Fanuc TP program (LS listing): _bgl_btn_pick.ls

/PROG  _BGL_BTN_PICK
/ATTR
OWNER		= MNEDITOR;
COMMENT		= "";
PROG_SIZE	= 225;
CREATE		= DATE 00-01-12  TIME 18:35:34;
MODIFIED	= DATE 00-01-12  TIME 18:35:34;
FILE_NAME	= ;
VERSION		= 0;
LINE_COUNT	= 4;
MEMORY_SIZE	= 581;
PROTECT		= READ_WRITE;
TCD:  STACK_SIZE	= 0,
      TASK_PRIORITY	= 50,
      TIME_SLICE	= 0,
      BUSY_LAMP_OFF	= 0,
      ABORT_REQUEST	= 0,
      PAUSE_REQUEST	= 0;
DEFAULT_GROUP	= *,*,*,*,*;
CONTROL_CODE	= 00000000 00000000;
LOCAL_REGISTERS	= 0,0,0;
/APPL
/APPL

AUTO_SINGULARITY_HEADER;
  ENABLE_SINGULARITY_AVOIDANCE   : FALSE;
/MN
   1:  IF (DI[103:PICK]) THEN ;
   2:  R[185:btnPickPressed]=1    ;
   3:  DO[106:TIMER STOP]=ON ;
   4:  ENDIF ;
/POS
/END
